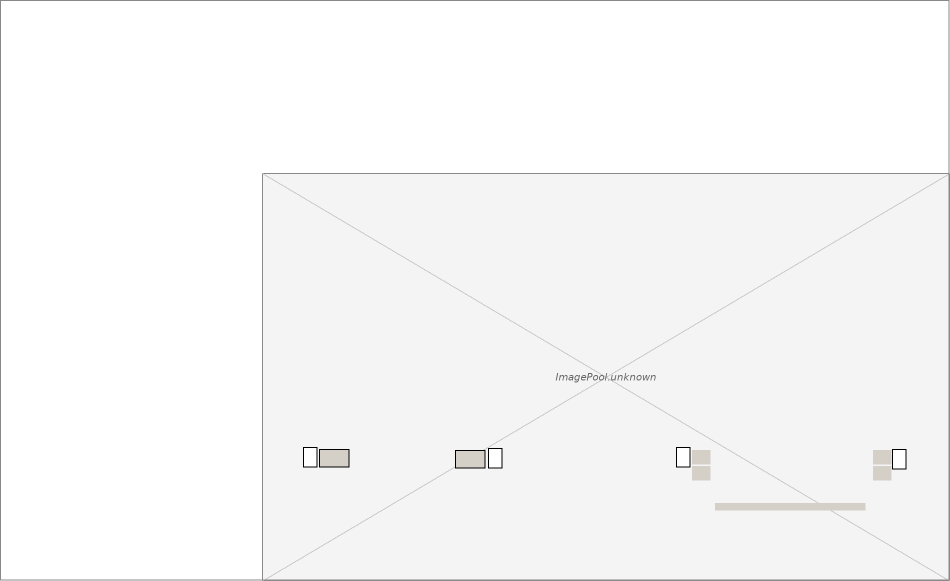
VISUALIZATION Visualization  // 950x581
    Image (262,173 688x408), image: ImagePool.unknown
    RoundedRectangle (488,448 14x20), colour toggle: MAIN.BlinkerLeft
    RoundedRectangle (303,447 14x20), colour toggle: MAIN.BlinkerRight
    RoundedRectangle (455,450 30x18), colour toggle: MAIN.LightsFront
    RoundedRectangle (676,447 14x20), colour toggle: MAIN.BlinkerLeft
    RoundedRectangle (892,449 14x20), colour toggle: MAIN.BlinkerRight
    RoundedRectangle (319,449 30x18), colour toggle: MAIN.LightsFront
    RoundedRectangle (692,450 18x14), colour toggle: MAIN.LightsRear
    RoundedRectangle (692,466 18x14), colour toggle: MAIN.LightsBrake
    RoundedRectangle (873,450 18x14), colour toggle: MAIN.LightsRear
    RoundedRectangle (873,466 18x14), colour toggle: MAIN.LightsBrake
    RoundedRectangle (715,503 150x7), colour toggle: MAIN.LightsReverse
END_VISUALIZATION

(* stored: Version 1.1.0.1, ProductVersion 3.1.4024.3
   Visu Visualization: Id {a493a650-b676-4b8f-b316-5c9c8526622b} *)
